PROGRAM MOVER
VAR
  nMover                : INT;

END_VAR



FOR nMover := 1 TO MAX_XPLANAR_MOVERS
DO
  fbMoverCtrl[nMover].MoverId   :=   TO_UINT(nMover);

  fbMoverCtrl[nMover].Ctrl      REF= MoverCtrl;
  fbMoverCtrl[nMover].State     REF= MoverState;
  fbMoverCtrl[nMover].MoveData  REF= MoveData;
  fbMoverCtrl[nMover].MoverInfo REF= MoverInfo[nMover];

  fbMoverCtrl[nMover].Mover     REF= MAIN.fbMover[nMover];
  fbMoverCtrl[nMover].Feedback  REF= MAIN.fbMoverFeedback[nMover];

  fbMoverCtrl[nMover]();
  fbMoverCtrl[nMover].Cycle();
END_FOR

END_PROGRAM

(* stored: Version 1.1.0.1, ProductVersion 3.1.4024.15
   POU MOVER: Id {2117d41c-bb68-4bc0-84d4-31f77add53d1}, SpecialFunc None *)
